(* CODESYS project RGB_CONTROL.project

Project tree, tasks and I/O mapping:
  Device : CECC-S, Festo AG & Co. KG, order no. 574416, version 3.5.7.27
    application Application
      libraries: Standard, * (System); Util, * (System); Network, 3.5.7.0 (3S - Smart Software Solutions GmbH); iParServer, * (3S - Smart Software Solutions GmbH); CommFB, * (3S - Smart Software Solutions GmbH); Festo_CECC_3, * (Festo AG & Co. KG)
      task MainTask (cyclic, interval t#20ms, priority 20) calls PLC_PRG
      task mem_clock (cyclic, interval t#50ms, priority 10) calls clk
      program PLC_PRG [ST]
      program clk [ST]
      global variables GVL
      function RGB_ [ST]
      function STR_TO_WORDS [ST]
      data type RGB_DATA
      function RGB [ST]
      data type RGB_UNION
    Onboard : CECC 14I/8O, Festo AG & Co. KG, version 3.4.5.5
        unmapped channels: Onboard Input, Onboard Output
      Digital Inputs
          unmapped channels: Onboard Input
      Digital Outputs
          unmapped channels: Onboard Output
    Ethernet : Ethernet, 3S - Smart Software Solutions GmbH, version 3.5.7.0
        settings: IPAddress = [10,0,0,121]; SubnetMask = [255,255,255,0]; GatewayAddress = [10,0,0,2]; NetworkInterfaceName = 'eth0'; NetworkInterfaceName = "eth0"
      Modbus_TCP_Master : Modbus TCP Master, 3S - Smart Software Solutions GmbH, version 3.5.6.0
          settings: AutoReconnect = TRUE
        Modbus_TCP_Slave_1 : Modbus TCP Slave, 3S - Smart Software Solutions GmbH, version 3.5.7.0
            settings: 16#0000 (=0).Function Code = 16; 16#0000 (=0).Write Offset = 0; 16#0000 (=0).Write Length = 4; 16#0000 (=0).Init Value = 10; Unit-ID = 1; IPAddress = [10, 0, 0, 49]; Read03.Function Code = 3; Read03.Read Offset = 16#0000; Read03.Read Length = 28; Read03.Write Offset = 0; Read03.Write Length = 0; Read03.Cycle Time = 1000; Read03.EnableRegisterBitMapping = FALSE; Shape.Function Code = 16; Shape.Read Offset = 0; Shape.Read Length = 0; Shape.Write Offset = 16#0004; Shape.Write Length = 4; Shape.Cycle Time = 100; Shape.EnableRegisterBitMapping = FALSE; Bitmap.Function Code = 16; Bitmap.Read Offset = 0; Bitmap.Read Length = 0; Bitmap.Write Offset = 16#0008; Bitmap.Write Length = 2; Bitmap.Cycle Time = 1000; Bitmap.EnableRegisterBitMapping = FALSE; Fill.Function Code = 16; Fill.Read Offset = 0; Fill.Read Length = 0; Fill.Write Offset = 16#001A; Fill.Write Length = 2; Fill.Cycle Time = 100; Rotate.Function Code = 16; Rotate.Read Offset = 0; Rotate.Read Length = 0; Rotate.Write Offset = 16#0018; Rotate.Write Length = 2; Rotate.Cycle Time = 100; TextSetup.Function Code = 16;
              TextSetup.Read Offset = 0; TextSetup.Read Length = 0; TextSetup.Write Offset = 16#000C; TextSetup.Write Length = 3; TextSetup.Cycle Time = 100; Font.Function Code = 6; Font.Read Offset = 0; Font.Read Length = 0; Font.Write Offset = 16#000F; Font.Write Length = 1; Font.Cycle Time = 100; Border.Function Code = 16; Border.Read Offset = 0; Border.Read Length = 0; Border.Write Offset = 16#000A; Border.Write Length = 2; Border.Cycle Time = 100; FloatValue_Setup.Function Code = 16; FloatValue_Setup.Read Offset = 0; FloatValue_Setup.Read Length = 0; FloatValue_Setup.Write Offset = 16#0010; FloatValue_Setup.Write Length = 8; FloatValue_Setup.Cycle Time = 100; FloatValue.Function Code = 16; FloatValue.Read Offset = 0; FloatValue.Read Length = 0; FloatValue.Write Offset = 16#0050; FloatValue.Write Length = 2; FloatValue.Cycle Time = 100; Text.Function Code = 16; Text.Read Offset = 0; Text.Read Length = 0; Text.Write Offset = 16#001E; Text.Write Length = 30; Text.Cycle Time = 100
            input  Application.PLC_PRG.rgb[0].REG_MAP AT %IW1 : ARRAY[0..27] OF WORD  // Read03
            output Application.PLC_PRG.rgb[0].rgb_bits.b0 AT %QX2.0 : BIT  // Shape
            output Application.PLC_PRG.rgb[0].shape : ARRAY[0..3] OF WORD  // Shape
            output Application.PLC_PRG.rgb[0].rgb_bits.b1 : BIT  // Bitmap
            output Application.PLC_PRG.rgb[0].bitmap AT %QW7 : ARRAY[0..1] OF WORD  // Bitmap
            output Application.PLC_PRG.rgb[0].rgb_bits.b2 : BIT  // Fill
            output Application.PLC_PRG.rgb[0].fill : ARRAY[0..1] OF WORD  // Fill
            output Application.PLC_PRG.rgb[0].rgb_bits.b3 : BIT  // Rotate
            output Application.PLC_PRG.rgb[0].rotate : ARRAY[0..1] OF WORD  // Rotate
            output Application.PLC_PRG.rgb[0].rgb_bits.b4 : BIT  // TextSetup
            output Application.PLC_PRG.rgb[0].text_set : ARRAY[0..2] OF WORD  // TextSetup
            output Application.PLC_PRG.rgb[0].rgb_bits.b5 : BIT  // Font
            output Application.PLC_PRG.rgb[0].font : ARRAY[0..0] OF WORD  // Font
            output Application.PLC_PRG.rgb[0].rgb_bits.b6 : BIT  // Border
            output Application.PLC_PRG.rgb[0].border : ARRAY[0..1] OF WORD  // Border
            output Application.PLC_PRG.rgb[0].rgb_bits.b7 : BIT  // FloatValue_Setup
            output Application.PLC_PRG.rgb[0].float_set : ARRAY[0..7] OF WORD  // FloatValue_Setup
            output Application.PLC_PRG.rgb[0].rgb_bits.b10 : BIT  // FloatValue
            output Application.PLC_PRG.rgb[0].floatV : ARRAY[0..1] OF WORD  // FloatValue
            output Application.PLC_PRG.rgb[0].rgb_bits.b11 : BIT  // Text
            output Application.PLC_PRG.rgb[0].textG : ARRAY[0..29] OF WORD  // Text
*)

// Device/Application/RGB_DATA
TYPE RGB_DATA :
STRUCT
	// Control bits 
	rgb_bits: RGB_UNION;
	
	// Register map
	REG_MAP: ARRAY[0..28] OF WORD; //x,y,xe,ye,s,sq,sw,sc,
	
	// Shape pos.   [0] {x start.}
	//				[1] {y start.}
	//				[2] {x finnish.}
	//				[3] {y finnish.}					
	shape_conf: ARRAY[0..3] OF WORD:=[0,10,10,10];
	// Shape set up [0] {0 = rect, 1 = triangle, 2 = circle, 3 = Straight kine, 4 = configured line}
	//				[1] {Quantity of shape around screen.}
	//				[2] {Weight of shape lines.}
	//				[3] {Color of shape.}
	shape: ARRAY[0..3] OF WORD:=[0,6,3,2016];
	
	// Run a bitmap [0] {Bitmap number.}
	//				[1] {Bitmap quantity.}
	bitmap: ARRAY[0..1] OF WORD:=[0,3];
	
	// Fill screen	[0] {0= no fill, 1= fill}
	//				[1] {Colour to fill.}
	fill: ARRAY[0..1] OF WORD:=[1,63488];
	
	// Rotation		[0] {0= no rotate, 1= rotate}
	//				[1]	{rotation speed.}
	rotate:ARRAY[0..1]OF WORD:=[1,10];
	
	// Show a border [0] {0= no border, 1= show border}
	//				 [1] {1= border width.}
	border:ARRAY[0..1]OF WORD:=[5,31];	
	
	// Text Pos		[0] {x position start}
	//				[1] {y position start}
	//				[2] {text color.}
	text_set:ARRAY[0..2]OF WORD:=[0,10,2016]; //x,y,col
	textG:ARRAY[0..29]OF WORD;
	
	font:WORD:=0;	
	float_set:ARRAY[0..7]OF WORD:=[0,1,0,100,10,90,31,63488];
	floatV:ARRAY[0..1]OF WORD;
	
END_STRUCT
END_TYPE

// Device/Application/RGB_UNION
TYPE RGB_UNION :
UNION
	b0: BOOL;
	b1: BOOL;
	b2: BOOL;
	b3: BOOL;
	b4: BOOL;
	b5: BOOL;
	b6: BOOL;
	b7: BOOL;
	b10: BOOL;
	b11: BOOL;
	b12: BOOL;
	b13: BOOL;
	b14: BOOL;
	b15: BOOL;
	b16: BOOL;
	b17: BOOL;
	
	inByte:  ARRAY[0..1] OF BYTE;
	
	inWord: WORD;
	
END_UNION
END_TYPE

// Device/Application/GVL
VAR_GLOBAL
	
	// Global mappings
	mclk: DWORD;
	
	// Display 1 mappings
(*	conf: ARRAY[0..28] OF WORD; //x,y,xe,ye,s,sq,sw,sc,
	shape_conf: ARRAY[0..3] OF WORD:=[0,10,10,10];
	shape: ARRAY[0..3] OF WORD:=[0,6,3,2016];
	bitmap: ARRAY[0..1] OF WORD:=[0,3];
	fill: ARRAY[0..1] OF WORD:=[1,63488];
	rotate:ARRAY[0..1]OF WORD:=[1,10];
	border:ARRAY[0..1]OF WORD:=[5,31];
	
	
	text_set:ARRAY[0..2]OF WORD:=[0,10,2016]; //x,y,col
	textG:ARRAY[0..29]OF WORD;
	font:WORD:=0;
	
	float_set:ARRAY[0..7]OF WORD:=[0,1,0,100,10,90,31,63488];
	floatV:ARRAY[0..1]OF WORD;
	*)
    cycle_display: BOOL;
	inputByte: BYTE;
	

	
	
	
	
END_VAR

// Device/Application/PLC_PRG
PROGRAM PLC_PRG
VAR
// lOCAL
 set_screen: BOOL;
// conf:BOOL;
//  set_shape: BOOL;
//  set_bitmap:BOOL;
//  fill_screen:BOOL;
//  b_rotate:BOOL;
// text_setup:BOOL;
//  font_change:BOOL;
//  borderset:BOOL;
//  border_toggle: BOOL;
//  rotate_toggle: BOOL;
//  last_border:WORD;
//  last_rotate: WORD;
//  textsend:BOOL;
  
//  float_setup:BOOL;
//  float_send:BOOL;

rgb: ARRAY[0..1] OF RGB_DATA;
  
T0: TON;
T1: TON;
T2: TON;

R0: R_TRIG;
R1: R_TRIG;


END_VAR


R0(CLK:=%IX0.3);
R1(CLK:= %IX0.6);
T0(IN:=set_screen,PT:=T#100MS);

cycle_display S= %IX0.7;
cycle_display R= %IX0.0 OR %IX0.1 OR %IX0.2 OR %IX0.3 OR %IX0.4;

T1(IN:= cycle_display AND NOT T1.Q, PT:= T#500MS);


RGB_(ADR(rgb[0]),R0.Q,R1.Q);

END_PROGRAM

// Device/Application/clk
PROGRAM clk
VAR
END_VAR
VAR RETAIN
   ms100: INT:=0;
   ms250: INT:=0;
   ms500: INT:=0;
   ms750: INT:=0;
   ms1000: INT:=0;
   ms2500: INT:=0;
  
END_VAR

ms100:= ms100 + 1;
ms250:= ms250+1;
ms500:= ms500+1;
ms750:=ms750+1;
ms1000:= ms1000+1;
ms2500:= ms2500+1;

IF ms100 = 1 THEN
	ms100:= 0;
	mclk:= SWITCHBIT(mclk,0);
END_IF

IF ms250 = 4 THEN
	ms250:= 0;
	mclk:=SWITCHBIT(mclk,1);
END_IF

IF ms500 = 9 THEN
	ms500:= 0;
	mclk:=SWITCHBIT(mclk,2);
END_IF

IF ms750 = 13 THEN
	ms750:= 0;
	mclk:=SWITCHBIT(mclk,3);
END_IF

IF ms1000 = 18 THEN
	ms1000:= 0;
	mclk:=SWITCHBIT(mclk,4);
END_IF

IF ms2500 = 45 THEN
	ms2500:= 0;
	mclk:=SWITCHBIT(mclk,5);
END_IF


%QX0.0:= EXTRACT(mclk,0);
%QX0.1:= EXTRACT(mclk,1);
%QX0.2:= EXTRACT(mclk,2);
%QX0.3:= EXTRACT(mclk,3);
%QX0.4:= EXTRACT(mclk,4);
%QX0.5:= EXTRACT(mclk,5);

END_PROGRAM

// Device/Application/RGB_
FUNCTION RGB_ : WORD
VAR_INPUT
	rgb:POINTER TO RGB_DATA;
	R0: BOOL;
	R1: BOOL;
END_VAR

// stack vars
VAR
END_VAR

// add to ram not stack
VAR_STAT

border_toggle: BOOL;
rotate_toggle: BOOL;
last_border: WORD;	
last_rotate: WORD;

END_VAR



// set toggle bits to send via modbus
IF (rgb^.rgb_bits.b0 OR rgb^.rgb_bits.b1 OR rgb^.rgb_bits.b2 OR rgb^.rgb_bits.b3 OR rgb^.rgb_bits.b4 OR rgb^.rgb_bits.b5 OR rgb^.rgb_bits.b6 
	OR rgb^.rgb_bits.b7 OR rgb^.rgb_bits.b10 OR rgb^.rgb_bits.b11 OR rgb^.rgb_bits.b12 OR rgb^.rgb_bits.b13 OR rgb^.rgb_bits.b14 OR rgb^.rgb_bits.b15)
	AND NOT rgb^.rgb_bits.b16 THEN
	rgb^.rgb_bits.b16 := TRUE;
END_IF

IF (rgb^.rgb_bits.b0 OR rgb^.rgb_bits.b1 OR rgb^.rgb_bits.b2 OR rgb^.rgb_bits.b3 OR rgb^.rgb_bits.b4 OR rgb^.rgb_bits.b5 OR rgb^.rgb_bits.b6 
	OR rgb^.rgb_bits.b7 OR rgb^.rgb_bits.b10 OR rgb^.rgb_bits.b11 OR rgb^.rgb_bits.b12 OR rgb^.rgb_bits.b13 OR rgb^.rgb_bits.b14 OR rgb^.rgb_bits.b15)
	AND rgb^.rgb_bits.b16 AND  rgb^.rgb_bits.b17  THEN
	rgb^.rgb_bits.b17 := FALSE;
END_IF


IF %IX0.0  THEN
	rgb^.textG:= STR_TO_WORDS('Hello!!',0,1);
	rgb^.rgb_bits.b11:= TRUE;
ELSIF %IX0.1  THEN
	rgb^.rgb_bits.b1:= TRUE;  //bitmap
ELSIF %IX0.2  THEN	
	rgb^.rgb_bits.b0 := true; //set_shape
ELSIF R0 THEN
	border_toggle:= NOT border_toggle;
	IF border_toggle THEN
		last_border:= rgb^.border[0];
		rgb^.border[0]:= 0;
	ELSE
		rgb^.border[0]:= last_border;
	END_IF
	rgb^.rgb_bits.b6 := true;  //borderset;
ELSIF %IX0.4 THEN
	rgb^.rgb_bits.b2 := true;  //fill_screen
ELSIF R1 THEN
	rotate_toggle := NOT rotate_toggle;
	IF rotate_toggle THEN
		last_rotate := rgb^.rotate[1];
		rgb^.rotate[1] := 0;
	ELSE
		rgb^.rotate[1] := last_rotate;
	END_IF
	rgb^.rgb_bits.b3 := true ;   //b_rotate;

END_IF;

END_FUNCTION

// Device/Application/RGB
FUNCTION RGB : WORD
VAR_INPUT

// rgb_data: Pointer to RGB_DATA;

END_VAR
VAR
bitx: BOOL;
err: word;
END_VAR


bitx := TRUE;



//IF (set_shape OR set_bitmap OR fill_screen OR conf OR b_rotate OR text_setup OR font_change OR borderset OR textsend)AND NOT set_screen THEN
//	set_screen:= TRUE;
//END_IF;
	
//IF (set_shape OR set_bitmap OR fill_screen OR conf OR b_rotate OR text_setup OR font_change OR borderset OR textsend) AND set_screen AND T0.Q THEN	
//	set_screen:= fill_screen:= conf:= set_bitmap:= set_shape:= b_rotate:= text_setup:= font_change:= borderset:= textsend:= FALSE;
//END_IF

(*
IF rgb_bits.b0 AND cycle_display THEN
	inputByte := ROL(inputByte,1);
	IF inputByte >= 32  THEN
		inputByte := 1;	
    ELSIF inputByte = 0 THEN
		inputByte := 1;	
	END_IF	
END_IF

IF NOT cycle_display THEN
	inputByte := 0;
END_IF

IF %IX0.0 OR inputByte = 1 THEN
	textG:= STR_TO_WORDS('Hello!!',0,1);
	textsend:= TRUE;
ELSIF %IX0.1 OR inputByte = 2 THEN
	set_bitmap:= TRUE;
ELSIF %IX0.2 OR inputByte = 4 THEN	
	set_shape:= TRUE;
ELSIF R0.Q THEN
	border_toggle:= NOT border_toggle;
	IF border_toggle THEN
		last_border:= border[0];
		border[0]:= 0;
	ELSE
		border[0]:= last_border;
	END_IF
	borderset:= TRUE;
ELSIF %IX0.4 OR inputByte = 16 THEN
	fill_screen:= TRUE;
ELSIF R1.Q THEN
	rotate_toggle := NOT rotate_toggle;
	IF rotate_toggle THEN
		last_rotate := rotate[1];
		rotate[1] := 0;
	ELSE
		rotate[1] := last_rotate;
	END_IF
	b_rotate := TRUE;

END_IF;*)

END_FUNCTION

// Device/Application/STR_TO_WORDS
FUNCTION STR_TO_WORDS : ARRAY[0..29]OF WORD
VAR_INPUT
 text:  STRING(60);
 pos:   INT;
 byte_order:INT:=0;
	
END_VAR
VAR
Char: POINTER TO BYTE;
indx: INT;
byt: ARRAY[0..1] OF BYTE;
wIndx:INT:= 0;
	
		
END_VAR



Char:= ADR(text);
wIndx:= 0;

FOR indx:=POS TO LEN(text) BY 2 DO

	byt[0]:= Char^;	
	Char:= Char+1;
	byt[1]:= Char^;
	Char:= Char + 1;	

	IF byte_order = 0 THEN
		STR_TO_WORDS[wIndx] := BYTE_TO_WORD(byt[1]);
		STR_TO_WORDS[wIndx]:= ROL(STR_TO_WORDS[wIndx],8);
		STR_TO_WORDS[wIndx]:= STR_TO_WORDS[wIndx] +  BYTE_TO_WORD(byt[0]);
	ELSE
		STR_TO_WORDS[wIndx] := BYTE_TO_WORD(byt[0]);
		STR_TO_WORDS[wIndx]:= ROL(STR_TO_WORDS[wIndx],8);
		STR_TO_WORDS[wIndx]:= STR_TO_WORDS[wIndx] +  BYTE_TO_WORD(byt[1]);		
	END_IF
	wIndx:= wIndx + 1;
END_FOR

END_FUNCTION
